(* PLC project PLC1, Unknown Unnamed 1 *)
(* stored: creationDateTime 2021-02-24T14:42:08, modificationDateTime 2024-08-06T14:57:46 *)

PROGRAM PLC3
  VAR_INPUT
    level : DINT;
  END_VAR
  VAR_OUTPUT
    pump : BOOL;
  END_VAR
  VAR
    low : BOOL;
    high : BOOL;
    low_3 : DINT := 0;
    high_3 : DINT := 10;
  END_VAR

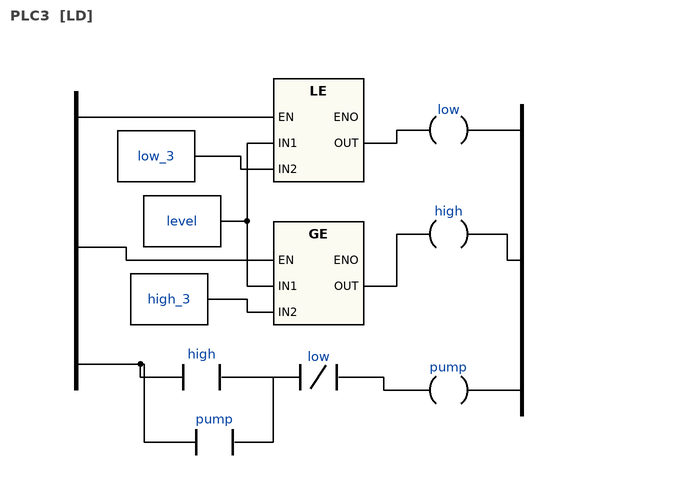
(* LD diagram, written out as Structured Text *)
high := level >= high_3;
low := level <= low_3;
pump := (high OR pump) AND NOT low;
END_PROGRAM

PROGRAM PLC2
  VAR_INPUT
    level : DINT;
  END_VAR
  VAR_OUTPUT
    request : BOOL;
  END_VAR
  VAR
    open_req : BOOL;
    close_req : BOOL;
    low_2 : DINT := 10;
    high_2 : DINT := 20;
  END_VAR

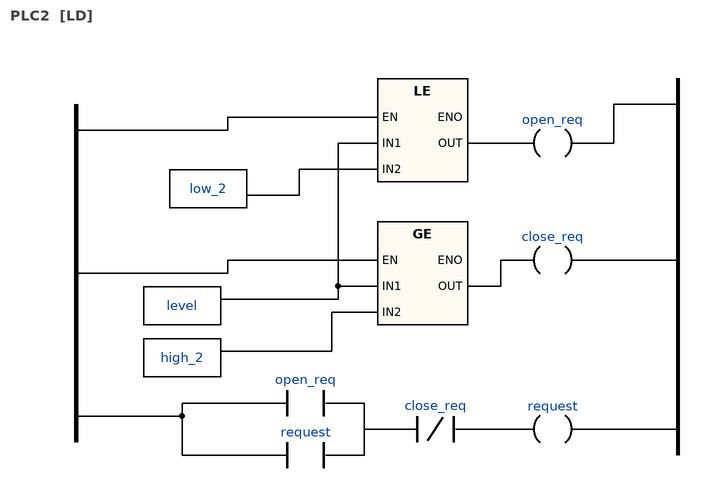
(* LD diagram, written out as Structured Text *)
close_req := level >= high_2;
open_req := level <= low_2;
request := (open_req OR request) AND NOT close_req;
END_PROGRAM

FUNCTION_BLOCK check_pumps
  VAR_INPUT
    IN1 : DINT;
    IN2 : DINT;
  END_VAR
  VAR_OUTPUT
    OUT : BOOL;
  END_VAR
  VAR
    i : INT;
  END_VAR

            if IN1 < IN2 then
  OUT:=TRUE;
end_if;
if IN1 >= IN2 then
  OUT:= FALSE;
end_if;

i:=0;
while i< 4 do
    OUT:=FALSE;
end_while;

          
END_FUNCTION_BLOCK

FUNCTION_BLOCK value_filtering
  VAR_INPUT
    IN1 : DINT;
  END_VAR
  VAR_OUTPUT
    real_value : DINT;
  END_VAR
  VAR
    i : INT;
  END_VAR

            real_value := IN1 - 5;


          
END_FUNCTION_BLOCK

PROGRAM PLC1
  VAR_INPUT
    level : DINT;
    request : DINT;
  END_VAR
  VAR_OUTPUT
    pumps : BOOL;
    pumps_state : BOOL;
    valve : BOOL;
    real_value : DINT;
  END_VAR
  VAR
    low : BOOL;
    high : BOOL;
    open_req : BOOL;
    close_req : BOOL;
    low_1 : DINT := 40;
    high_1 : DINT := 80;
    value_filtering0 : value_filtering;
    check_pumps0 : check_pumps;
    TON0 : TON;
  END_VAR

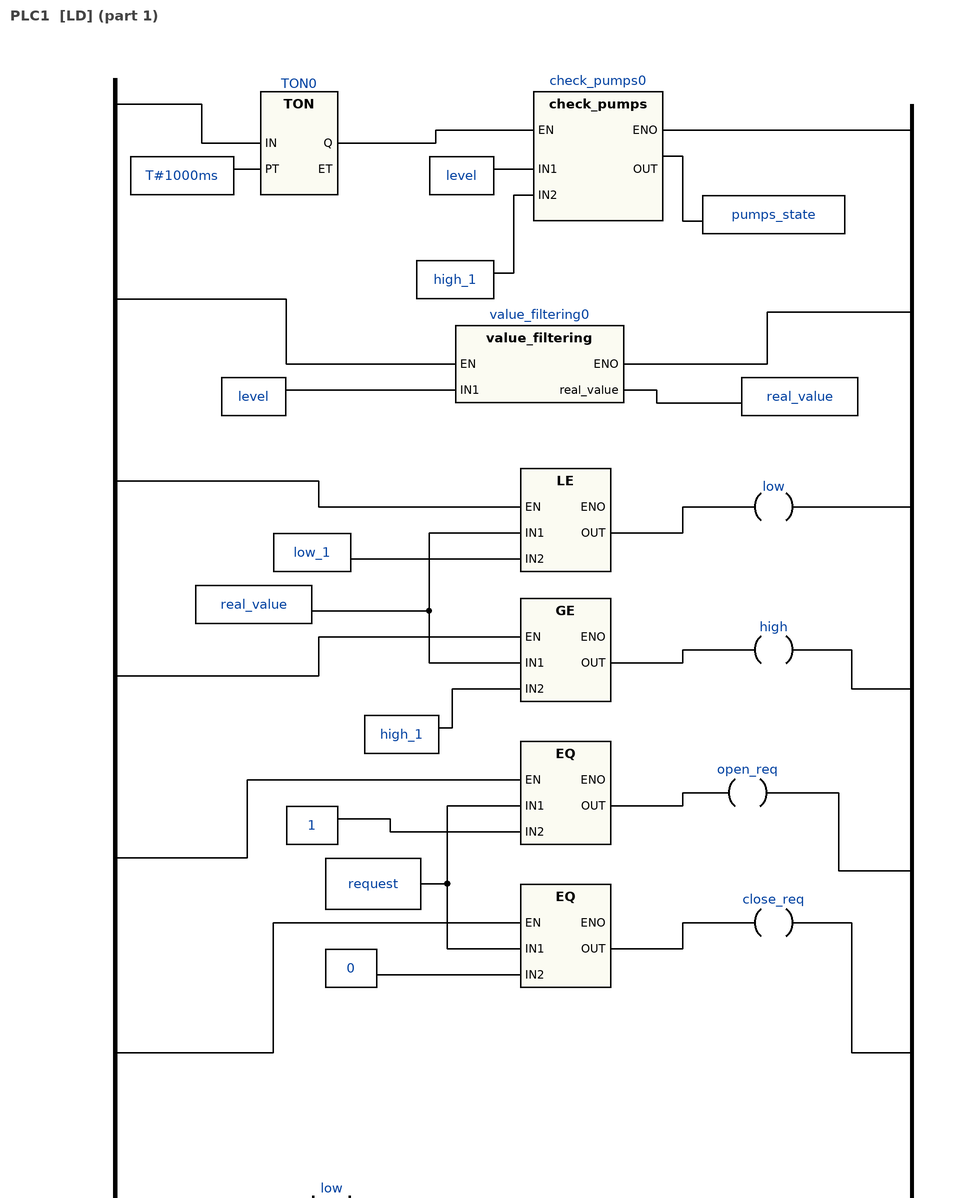
(* LD diagram, written out as Structured Text *)
low := real_value <= low_1;
high := real_value >= high_1;
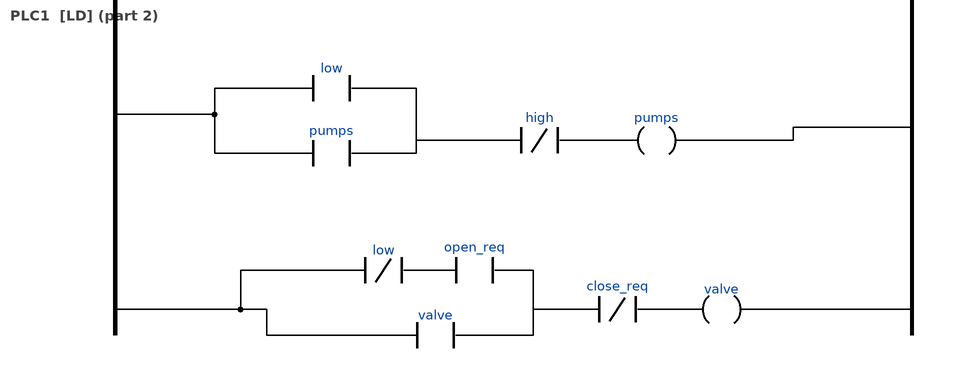
pumps := (low OR pumps) AND NOT high;
valve := (NOT low AND open_req OR valve) AND NOT close_req;
open_req := request = 1;
close_req := request = 0;
value_filtering0(IN1 := level);
real_value := value_filtering0.real_value;
TON0(IN := TRUE, PT := T#1000ms);
check_pumps0(EN := TON0.Q, IN1 := level, IN2 := high_1);
IF check_pumps0.ENO THEN pumps_state := check_pumps0.OUT; END_IF;
END_PROGRAM

CONFIGURATION Config0
  RESOURCE Res0 ON PLC
    TASK task0(INTERVAL := T#20ms, PRIORITY := 0);
    TASK task1(INTERVAL := T#20ms, PRIORITY := 0);
    TASK task2(INTERVAL := T#20ms, PRIORITY := 0);
    PROGRAM instance0 WITH task0 : PLC1;
    PROGRAM instance1 WITH task1 : PLC2;
    PROGRAM instance2 WITH task2 : PLC3;
  END_RESOURCE
END_CONFIGURATION
